
FUNCTION FC19 : VOID
//QTRANSN

VAR_INPUT
    IN1:REAL;
    IN2:REAL;
END_VAR

VAR_OUTPUT
    OUT:REAL;
END_VAR

    OUT:=IN1;
END_FUNCTION
